{attribute addProperty BoxType "EL3182-0000-0016"}
{attribute addProperty Id "StatusAT %I*Status_391E3AAC1621ValueAT %I*INT16217"}
{attribute addProperty CRC "3526367581"}
{attribute addProperty SizeInBites "32"}
{attribute addProperty SizeInBytes "4"}
TYPE Ch_2_Al_Inputs_D230195D :
STRUCT
	{attribute addProperty Name "Status"}
	Status AT %I* : Status_391E3AAC;
	{attribute addProperty Name "Value"}
	Value AT %I* : INT;
END_STRUCT
END_TYPE

(* stored: Version 1.2.0.0, ProductVersion 3.1.4024.9
   DUT Ch_2_Al_Inputs_D230195D: Id {9f0ad71d-bc91-4a06-b88f-bf7d33009373} *)
